PROGRAM Safety
VAR
END_VAR

END_PROGRAM

(* stored: Version 1.1.0.1, ProductVersion 3.1.4024.12
   POU Safety: Id {e95ddaa8-e370-40ac-9dda-44ae81d8a2b4}, SpecialFunc None *)
